// SIMATIC S7-200 project (STEP 7-Micro/WIN), CPU 226 REL 01.23

ORGANIZATION_BLOCK MAIN:OB1
TITLE= 
// PROGRAM COMMENTS
// Press F1 for help and example program
//  
BEGIN
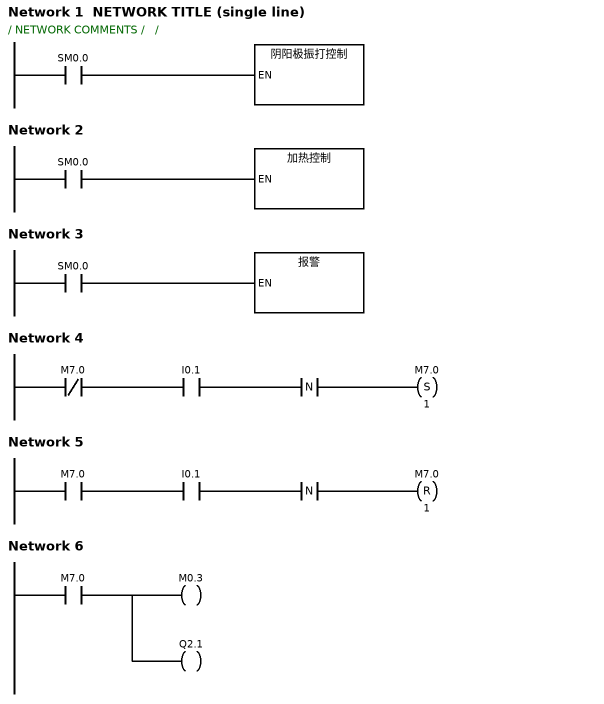
Network 1 // NETWORK TITLE (single line)
//  
// NETWORK COMMENTS
//  
// 
LD     SM0.0
CALL   阴阳极振打控制:SBR0
Network 2
LD     SM0.0
CALL   加热控制:SBR1
Network 3
LD     SM0.0
CALL   报警:SBR2
Network 4
LDN    M7.0
A      I0.1
ED
S      M7.0, 1
Network 5
LD     M7.0
A      I0.1
ED
R      M7.0, 1
Network 6
LD     M7.0
=      M0.3
=      Q2.1
END_ORGANIZATION_BLOCK

SUBROUTINE_BLOCK 阴阳极振打控制:SBR0
TITLE= 
// SUBROUTINE COMMENTS
// Press F1 for help and example program
//  
BEGIN
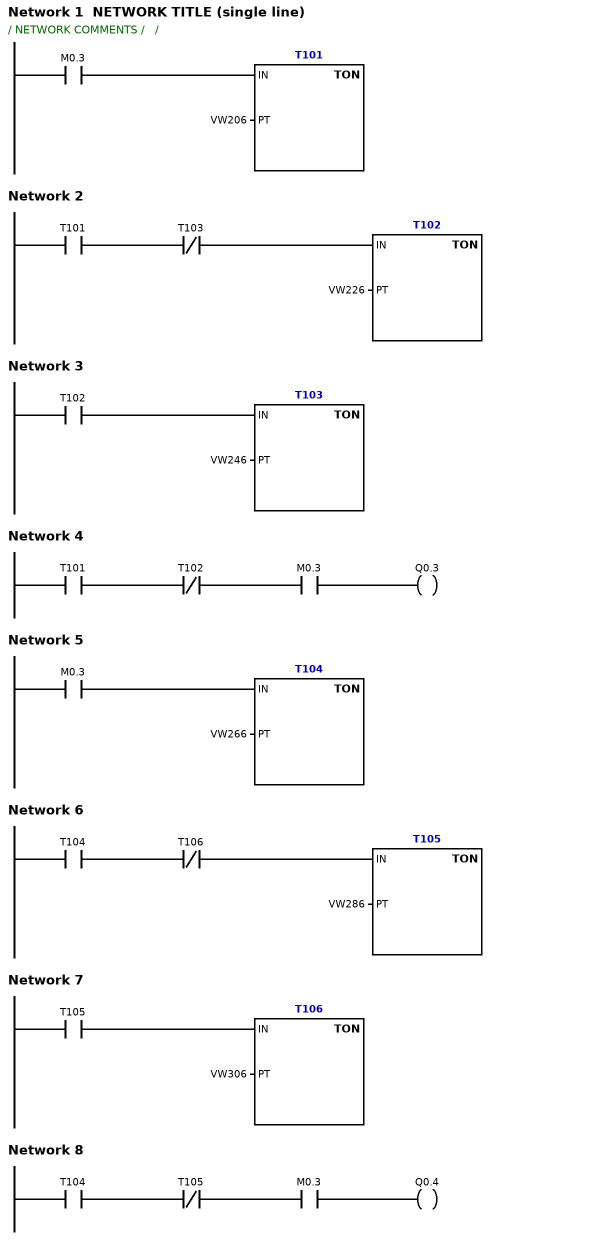
Network 1 // NETWORK TITLE (single line)
//  
// NETWORK COMMENTS
//  
// 
LD     M0.3
TON    T101, VW206
Network 2
LD     T101
AN     T103
TON    T102, VW226
Network 3
LD     T102
TON    T103, VW246
Network 4
LD     T101
AN     T102
A      M0.3
=      Q0.3
Network 5
LD     M0.3
TON    T104, VW266
Network 6
LD     T104
AN     T106
TON    T105, VW286
Network 7
LD     T105
TON    T106, VW306
Network 8
LD     T104
AN     T105
A      M0.3
=      Q0.4
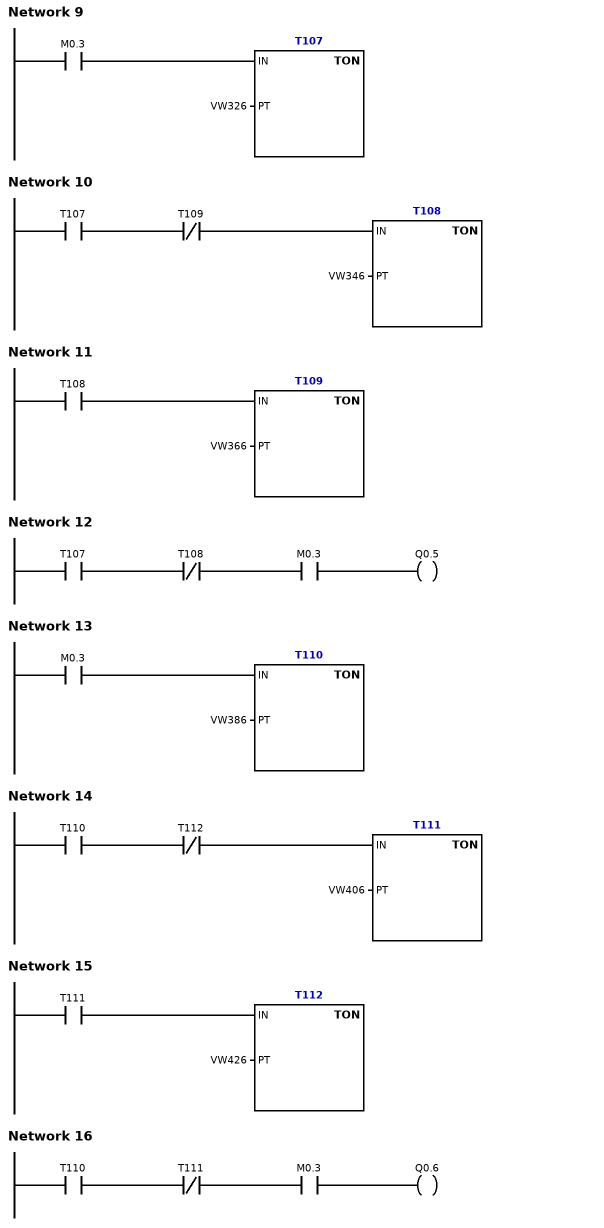
Network 9
LD     M0.3
TON    T107, VW326
Network 10
LD     T107
AN     T109
TON    T108, VW346
Network 11
LD     T108
TON    T109, VW366
Network 12
LD     T107
AN     T108
A      M0.3
=      Q0.5
Network 13
LD     M0.3
TON    T110, VW386
Network 14
LD     T110
AN     T112
TON    T111, VW406
Network 15
LD     T111
TON    T112, VW426
Network 16
LD     T110
AN     T111
A      M0.3
=      Q0.6
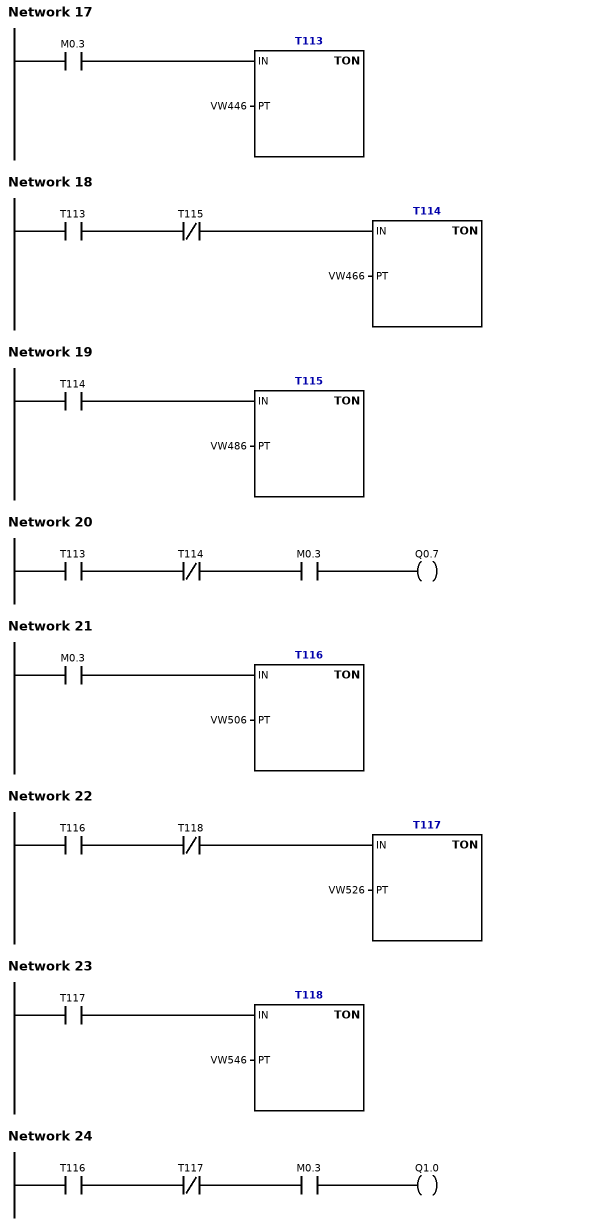
Network 17
LD     M0.3
TON    T113, VW446
Network 18
LD     T113
AN     T115
TON    T114, VW466
Network 19
LD     T114
TON    T115, VW486
Network 20
LD     T113
AN     T114
A      M0.3
=      Q0.7
Network 21
LD     M0.3
TON    T116, VW506
Network 22
LD     T116
AN     T118
TON    T117, VW526
Network 23
LD     T117
TON    T118, VW546
Network 24
LD     T116
AN     T117
A      M0.3
=      Q1.0
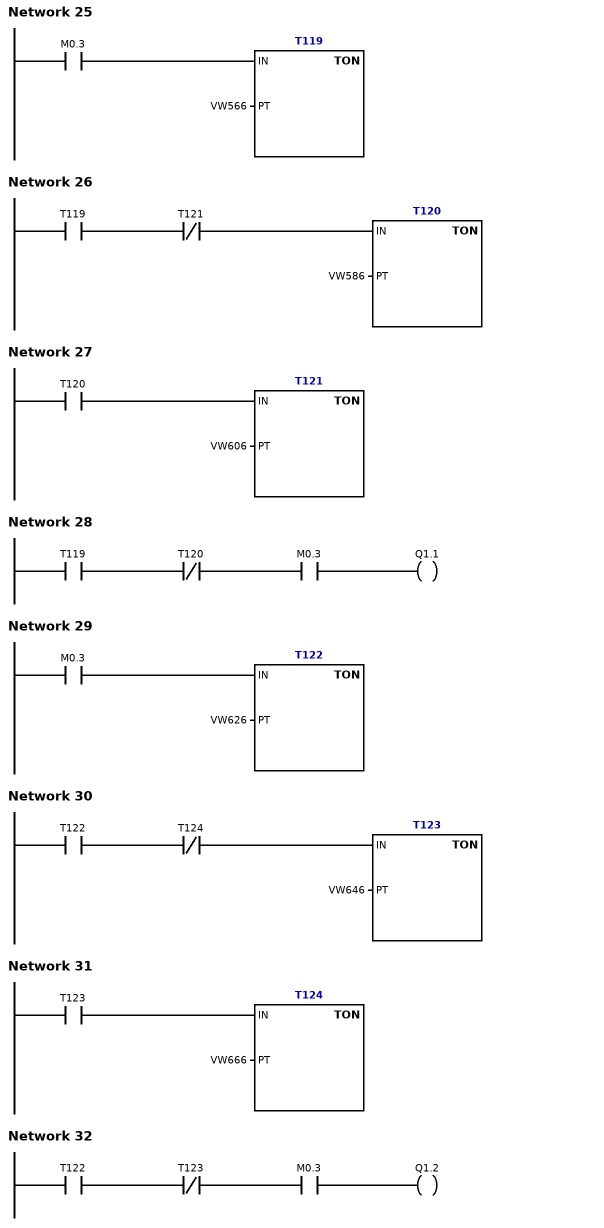
Network 25
LD     M0.3
TON    T119, VW566
Network 26
LD     T119
AN     T121
TON    T120, VW586
Network 27
LD     T120
TON    T121, VW606
Network 28
LD     T119
AN     T120
A      M0.3
=      Q1.1
Network 29
LD     M0.3
TON    T122, VW626
Network 30
LD     T122
AN     T124
TON    T123, VW646
Network 31
LD     T123
TON    T124, VW666
Network 32
LD     T122
AN     T123
A      M0.3
=      Q1.2
END_SUBROUTINE_BLOCK

SUBROUTINE_BLOCK 加热控制:SBR1
TITLE=
BEGIN
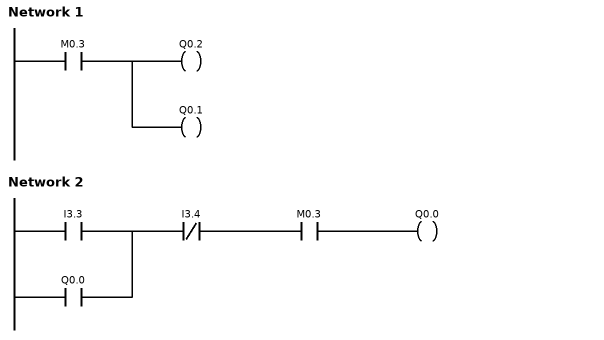
Network 1
LD     M0.3
=      Q0.2
=      Q0.1
Network 2
LD     I3.3
O      Q0.0
AN     I3.4
A      M0.3
=      Q0.0
END_SUBROUTINE_BLOCK

SUBROUTINE_BLOCK 报警:SBR2
TITLE=
BEGIN
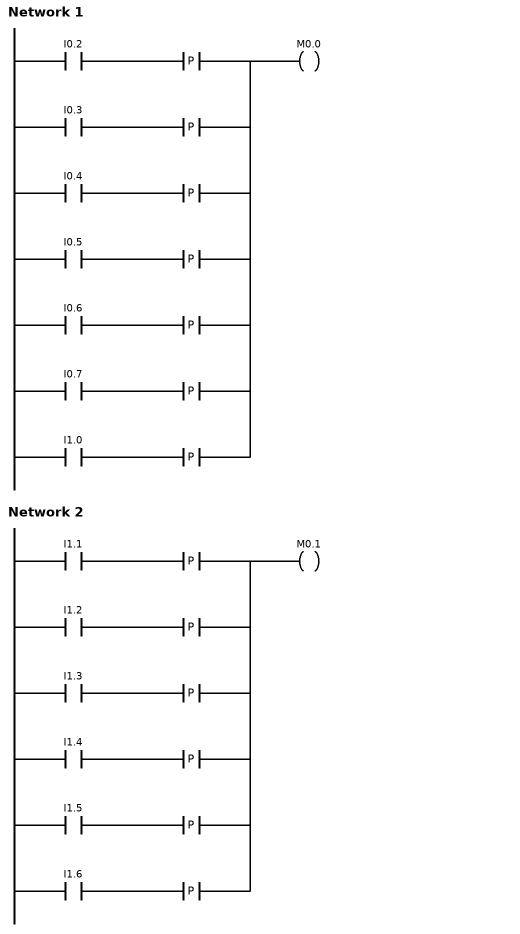
Network 1
LD     I0.2
EU
LD     I0.3
EU
OLD
LD     I0.4
EU
OLD
LD     I0.5
EU
OLD
LD     I0.6
EU
OLD
LD     I0.7
EU
OLD
LD     I1.0
EU
OLD
=      M0.0
Network 2
LD     I1.1
EU
LD     I1.2
EU
OLD
LD     I1.3
EU
OLD
LD     I1.4
EU
OLD
LD     I1.5
EU
OLD
LD     I1.6
EU
OLD
=      M0.1
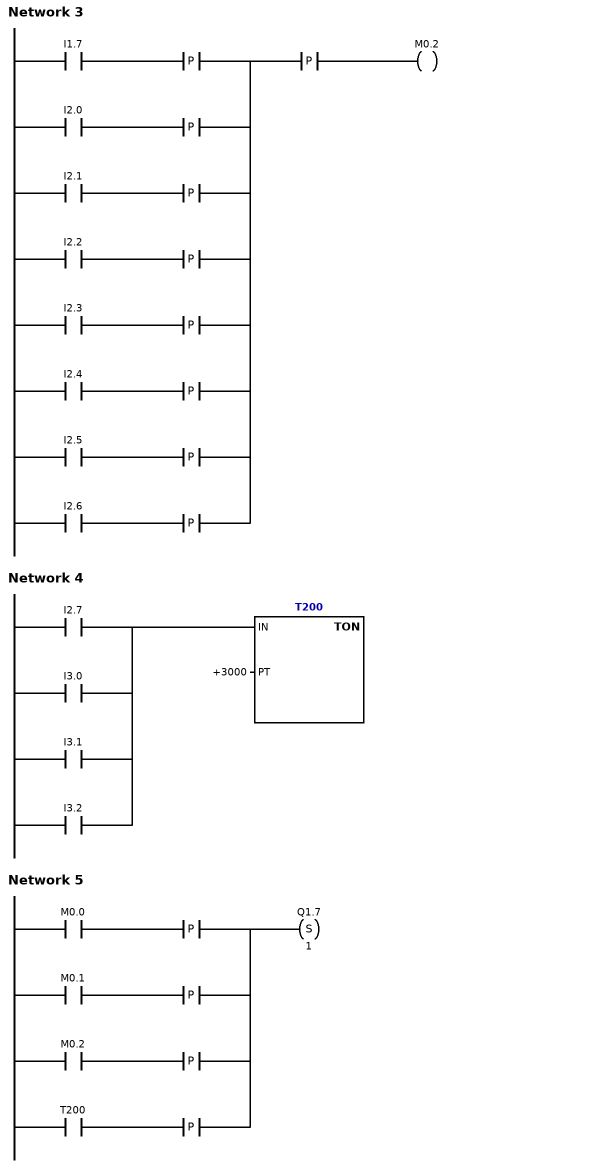
Network 3
LD     I1.7
EU
LD     I2.0
EU
OLD
LD     I2.1
EU
OLD
LD     I2.2
EU
OLD
LD     I2.3
EU
OLD
LD     I2.4
EU
OLD
LD     I2.5
EU
OLD
LD     I2.6
EU
OLD
EU
=      M0.2
Network 4
LD     I2.7
O      I3.0
O      I3.1
O      I3.2
TON    T200, +3000
Network 5
LD     M0.0
EU
LD     M0.1
EU
OLD
LD     M0.2
EU
OLD
LD     T200
EU
OLD
S      Q1.7, 1
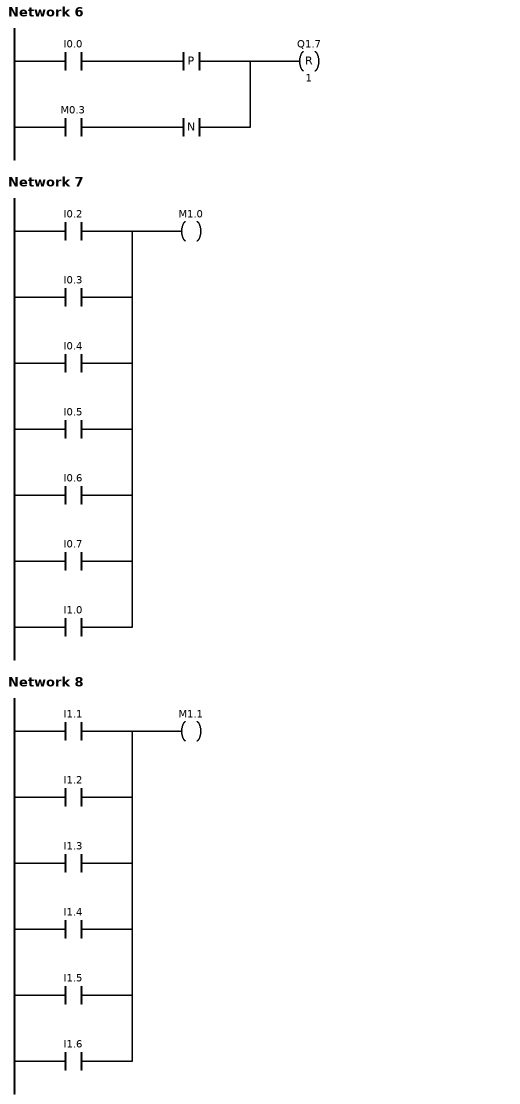
Network 6
LD     I0.0
EU
LD     M0.3
ED
OLD
R      Q1.7, 1
Network 7
LD     I0.2
O      I0.3
O      I0.4
O      I0.5
O      I0.6
O      I0.7
O      I1.0
=      M1.0
Network 8
LD     I1.1
O      I1.2
O      I1.3
O      I1.4
O      I1.5
O      I1.6
=      M1.1
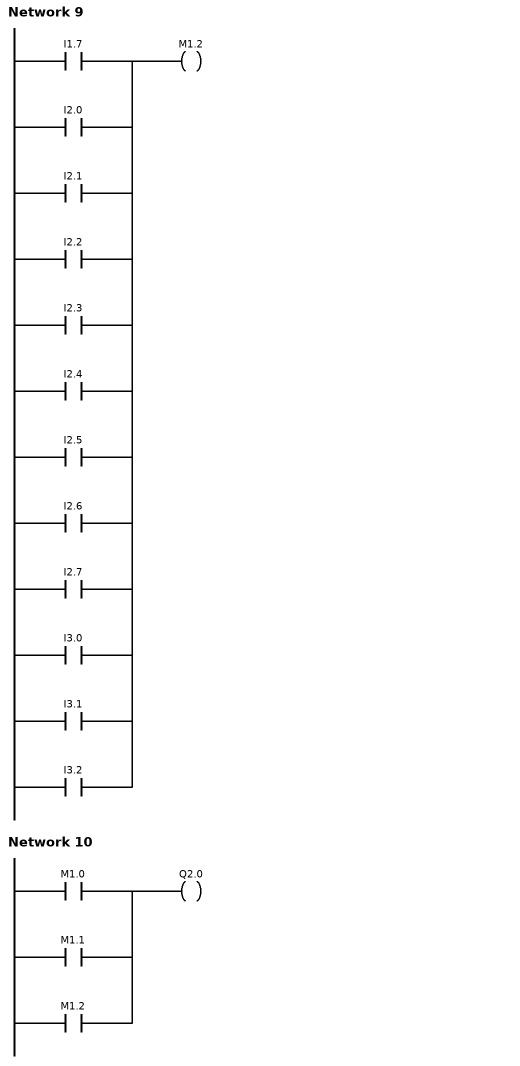
Network 9
LD     I1.7
O      I2.0
O      I2.1
O      I2.2
O      I2.3
O      I2.4
O      I2.5
O      I2.6
O      I2.7
O      I3.0
O      I3.1
O      I3.2
=      M1.2
Network 10
LD     M1.0
O      M1.1
O      M1.2
=      Q2.0
END_SUBROUTINE_BLOCK

DATA_BLOCK_TAB 用户定义1
BEGIN
VB0      16#0
VB1      16#0
VB2      16#0
VB3      16#0
VB4      16#0
VB5      16#0
VB6      16#0
VB7      16#0
VB8      16#0
VB9      16#0
VB10     16#0
VB11     16#0
VB12     16#0
VB13     16#0
VB14     16#0
VB15     16#0
VB16     16#0
VB17     16#0
VB18     16#0
VB19     16#0
VB20     16#0
VB21     16#0
VB22     16#0
VB23     16#0
VB24     16#0
VB25     16#0
VB26     16#0
VB27     16#0
VB28     16#0
VB29     16#0
VB30     16#0
VB31     16#0
VB32     16#0
VB33     16#0
VB34     16#0
VB35     16#0
VB36     16#0
VB37     16#0
VB38     16#0
VB39     16#0
VB40     16#0
VB41     16#0
VB42     16#0
VB43     16#0
VB44     16#0
VB45     16#0
VB46     16#0
VB47     16#0
VB48     16#0
VB49     16#0
VB50     16#0
VB51     16#0
VB52     16#0
VB53     16#0
VB54     16#0
VB55     16#0
VB56     16#0
VB57     16#0
VB58     16#0
VB59     16#0
VB60     16#0
VB61     16#0
VB62     16#0
VB63     16#0
VB64     16#0
VB65     16#0
VB66     16#0
VB67     16#0
VB68     16#0
VB69     16#0
VB70     16#0
VB71     16#0
VB72     16#0
VB73     16#0
VB74     16#0
VB75     16#0
VB76     16#0
VB77     16#0
VB78     16#0
VB79     16#0
VB80     16#0
VB81     16#0
VB82     16#0
VB83     16#0
VB84     16#0
VB85     16#0
VB86     16#0
VB87     16#0
VB88     16#0
VB89     16#0
VB90     16#0
VB91     16#0
VB92     16#0
VB93     16#0
VB94     16#0
VB95     16#0
VB96     16#0
VB97     16#0
VB98     16#0
VB99     16#0
VB100    16#0
VB101    16#0
VB102    16#0
VB103    16#0
VB104    16#0
VB105    16#0
VB106    16#0
VB107    16#0
VB108    16#0
VB109    16#0
VB110    16#0
VB111    16#0
VB112    16#0
VB113    16#0
VB114    16#0
VB115    16#0
VB116    16#0
VB117    16#0
VB118    16#0
VB119    16#0
VB120    16#0
VB121    16#0
VB122    16#0
VB123    16#0
VB124    16#0
VB125    16#0
VB126    16#0
VB127    16#0
VB128    16#0
VB129    16#0
VB130    16#0
VB131    16#0
VB132    16#0
VB133    16#0
VB134    16#0
VB135    16#0
VB136    16#0
VB137    16#0
VB138    16#0
VB139    16#0
VB140    16#0
VB141    16#0
VB142    16#0
VB143    16#0
VB144    16#0
VB145    16#0
VB146    16#0
VB147    16#0
VB148    16#0
VB149    16#0
VB150    16#0
VB151    16#0
VB152    16#0
VB153    16#0
VB154    16#0
VB155    16#0
VB156    16#0
VB157    16#0
VB158    16#0
VB159    16#0
VB160    16#0
VB161    16#0
VB162    16#0
VB163    16#0
VB164    16#0
VB165    16#0
VB166    16#0
VB167    16#0
VB168    16#0
VB169    16#0
VB170    16#0
VB171    16#0
VB172    16#0
VB173    16#0
VB174    16#0
VB175    16#0
VB176    16#0
VB177    16#0
VB178    16#0
VB179    16#0
VB180    16#0
VB181    16#0
VB182    16#0
VB183    16#0
VB184    16#0
VB185    16#0
VB186    16#0
VB187    16#0
VB188    16#0
VB189    16#0
VB190    16#0
VB191    16#0
VB192    16#0
VB193    16#0
VB194    16#0
VB195    16#0
VB196    16#0
VB197    16#0
VB198    16#0
VB199    16#0
VB200    16#0
VB201    16#0
VB202    16#0
VB203    16#0
VB204    16#0
VB205    16#0
VB206    16#0
VB207    16#0
VB208    16#0
VB209    16#0
VB210    16#0
VB211    16#0
VB212    16#0
VB213    16#0
VB214    16#0
VB215    16#0
VB216    16#0
VB217    16#0
VB218    16#0
VB219    16#0
VB220    16#0
VB221    16#0
VB222    16#0
VB223    16#0
VB224    16#0
VB225    16#0
VB226    16#5
VB227    16#DC
VB228    16#0
VB229    16#0
VB230    16#0
VB231    16#0
VB232    16#0
VB233    16#0
VB234    16#0
VB235    16#0
VB236    16#0
VB237    16#0
VB238    16#0
VB239    16#0
VB240    16#0
VB241    16#0
VB242    16#0
VB243    16#0
VB244    16#0
VB245    16#0
VB246    16#5
VB247    16#DC
VB248    16#0
VB249    16#0
VB250    16#0
VB251    16#0
VB252    16#0
VB253    16#0
VB254    16#0
VB255    16#0
VB256    16#0
VB257    16#0
VB258    16#0
VB259    16#0
VB260    16#0
VB261    16#0
VB262    16#0
VB263    16#0
VB264    16#0
VB265    16#0
VB266    16#5
VB267    16#DC
VB268    16#0
VB269    16#0
VB270    16#0
VB271    16#0
VB272    16#0
VB273    16#0
VB274    16#0
VB275    16#0
VB276    16#0
VB277    16#0
VB278    16#0
VB279    16#0
VB280    16#0
VB281    16#0
VB282    16#0
VB283    16#0
VB284    16#0
VB285    16#0
VB286    16#5
VB287    16#DC
VB288    16#0
VB289    16#0
VB290    16#0
VB291    16#0
VB292    16#0
VB293    16#0
VB294    16#0
VB295    16#0
VB296    16#0
VB297    16#0
VB298    16#0
VB299    16#0
VB300    16#0
VB301    16#0
VB302    16#0
VB303    16#0
VB304    16#0
VB305    16#0
VB306    16#11
VB307    16#94
VB308    16#0
VB309    16#0
VB310    16#0
VB311    16#0
VB312    16#0
VB313    16#0
VB314    16#0
VB315    16#0
VB316    16#0
VB317    16#0
VB318    16#0
VB319    16#0
VB320    16#0
VB321    16#0
VB322    16#0
VB323    16#0
VB324    16#0
VB325    16#0
VB326    16#11
VB327    16#94
VB328    16#0
VB329    16#0
VB330    16#0
VB331    16#0
VB332    16#0
VB333    16#0
VB334    16#0
VB335    16#0
VB336    16#0
VB337    16#0
VB338    16#0
VB339    16#0
VB340    16#0
VB341    16#0
VB342    16#0
VB343    16#0
VB344    16#0
VB345    16#0
VB346    16#5
VB347    16#DC
VB348    16#0
VB349    16#0
VB350    16#0
VB351    16#0
VB352    16#0
VB353    16#0
VB354    16#0
VB355    16#0
VB356    16#0
VB357    16#0
VB358    16#0
VB359    16#0
VB360    16#0
VB361    16#0
VB362    16#0
VB363    16#0
VB364    16#0
VB365    16#0
VB366    16#29
VB367    16#4
VB368    16#0
VB369    16#0
VB370    16#0
VB371    16#0
VB372    16#0
VB373    16#0
VB374    16#0
VB375    16#0
VB376    16#0
VB377    16#0
VB378    16#0
VB379    16#0
VB380    16#0
VB381    16#0
VB382    16#0
VB383    16#0
VB384    16#0
VB385    16#0
VB386    16#17
VB387    16#70
VB388    16#0
VB389    16#0
VB390    16#0
VB391    16#0
VB392    16#0
VB393    16#0
VB394    16#0
VB395    16#0
VB396    16#0
VB397    16#0
VB398    16#0
VB399    16#0
VB400    16#0
VB401    16#0
VB402    16#0
VB403    16#0
VB404    16#0
VB405    16#0
VB406    16#5
VB407    16#DC
VB408    16#0
VB409    16#0
VB410    16#0
VB411    16#0
VB412    16#0
VB413    16#0
VB414    16#0
VB415    16#0
VB416    16#0
VB417    16#0
VB418    16#0
VB419    16#0
VB420    16#0
VB421    16#0
VB422    16#0
VB423    16#0
VB424    16#0
VB425    16#0
VB426    16#40
VB427    16#74
VB428    16#0
VB429    16#0
VB430    16#0
VB431    16#0
VB432    16#0
VB433    16#0
VB434    16#0
VB435    16#0
VB436    16#0
VB437    16#0
VB438    16#0
VB439    16#0
VB440    16#0
VB441    16#0
VB442    16#0
VB443    16#0
VB444    16#0
VB445    16#0
VB446    16#5
VB447    16#DC
VB448    16#0
VB449    16#0
VB450    16#0
VB451    16#0
VB452    16#0
VB453    16#0
VB454    16#0
VB455    16#0
VB456    16#0
VB457    16#0
VB458    16#0
VB459    16#0
VB460    16#0
VB461    16#0
VB462    16#0
VB463    16#0
VB464    16#0
VB465    16#0
VB466    16#5
VB467    16#DC
VB468    16#0
VB469    16#0
VB470    16#0
VB471    16#0
VB472    16#0
VB473    16#0
VB474    16#0
VB475    16#0
VB476    16#0
VB477    16#0
VB478    16#0
VB479    16#0
VB480    16#0
VB481    16#0
VB482    16#0
VB483    16#0
VB484    16#0
VB485    16#0
VB486    16#5
VB487    16#DC
VB488    16#0
VB489    16#0
VB490    16#0
VB491    16#0
VB492    16#0
VB493    16#0
VB494    16#0
VB495    16#0
VB496    16#0
VB497    16#0
VB498    16#0
VB499    16#0
VB500    16#0
VB501    16#0
VB502    16#0
VB503    16#0
VB504    16#0
VB505    16#0
VB506    16#B
VB507    16#B8
VB508    16#0
VB509    16#0
VB510    16#0
VB511    16#0
VB512    16#0
VB513    16#0
VB514    16#0
VB515    16#0
VB516    16#0
VB517    16#0
VB518    16#0
VB519    16#0
VB520    16#0
VB521    16#0
VB522    16#0
VB523    16#0
VB524    16#0
VB525    16#0
VB526    16#5
VB527    16#DC
VB528    16#0
VB529    16#0
VB530    16#0
VB531    16#0
VB532    16#0
VB533    16#0
VB534    16#0
VB535    16#0
VB536    16#0
VB537    16#0
VB538    16#0
VB539    16#0
VB540    16#0
VB541    16#0
VB542    16#0
VB543    16#0
VB544    16#0
VB545    16#0
VB546    16#5
VB547    16#DC
VB548    16#0
VB549    16#0
VB550    16#0
VB551    16#0
VB552    16#0
VB553    16#0
VB554    16#0
VB555    16#0
VB556    16#0
VB557    16#0
VB558    16#0
VB559    16#0
VB560    16#0
VB561    16#0
VB562    16#0
VB563    16#0
VB564    16#0
VB565    16#0
VB566    16#11
VB567    16#94
VB568    16#0
VB569    16#0
VB570    16#0
VB571    16#0
VB572    16#0
VB573    16#0
VB574    16#0
VB575    16#0
VB576    16#0
VB577    16#0
VB578    16#0
VB579    16#0
VB580    16#0
VB581    16#0
VB582    16#0
VB583    16#0
VB584    16#0
VB585    16#0
VB586    16#5
VB587    16#DC
VB588    16#0
VB589    16#0
VB590    16#0
VB591    16#0
VB592    16#0
VB593    16#0
VB594    16#0
VB595    16#0
VB596    16#0
VB597    16#0
VB598    16#0
VB599    16#0
VB600    16#0
VB601    16#0
VB602    16#0
VB603    16#0
VB604    16#0
VB605    16#0
VB606    16#5
VB607    16#DC
VB608    16#0
VB609    16#0
VB610    16#0
VB611    16#0
VB612    16#0
VB613    16#0
VB614    16#0
VB615    16#0
VB616    16#0
VB617    16#0
VB618    16#0
VB619    16#0
VB620    16#0
VB621    16#0
VB622    16#0
VB623    16#0
VB624    16#0
VB625    16#0
VB626    16#17
VB627    16#70
VB628    16#0
VB629    16#0
VB630    16#0
VB631    16#0
VB632    16#0
VB633    16#0
VB634    16#0
VB635    16#0
VB636    16#0
VB637    16#0
VB638    16#0
VB639    16#0
VB640    16#0
VB641    16#0
VB642    16#0
VB643    16#0
VB644    16#0
VB645    16#0
VB646    16#5
VB647    16#DC
VB648    16#0
VB649    16#0
VB650    16#0
VB651    16#0
VB652    16#0
VB653    16#0
VB654    16#0
VB655    16#0
VB656    16#0
VB657    16#0
VB658    16#0
VB659    16#0
VB660    16#0
VB661    16#0
VB662    16#0
VB663    16#0
VB664    16#0
VB665    16#0
VB666    16#5
VB667    16#DC
VB668    16#0
VB669    16#0
VB670    16#0
VB671    16#0
VB672    16#0
VB673    16#0
VB674    16#0
VB675    16#0
VB676    16#0
VB677    16#0
VB678    16#0
VB679    16#0
VB680    16#0
VB681    16#0
VB682    16#0
VB683    16#0
VB684    16#0
VB685    16#0
VB686    16#B
VB687    16#B8
VB688    16#0
VB689    16#0
VB690    16#0
VB691    16#0
VB692    16#0
VB693    16#0
VB694    16#0
VB695    16#0
VB696    16#0
VB697    16#0
VB698    16#0
VB699    16#0
VB700    16#0
VB701    16#0
VB702    16#0
VB703    16#0
VB704    16#0
VB705    16#0
VB706    16#B
VB707    16#B8
VB708    16#0
VB709    16#0
VB710    16#0
VB711    16#0
VB712    16#0
VB713    16#0
VB714    16#0
VB715    16#0
VB716    16#0
VB717    16#0
VB718    16#0
VB719    16#0
VB720    16#0
VB721    16#0
VB722    16#0
VB723    16#0
VB724    16#0
VB725    16#0
VB726    16#B
VB727    16#B8
VB728    16#0
VB729    16#0
VB730    16#0
VB731    16#0
VB732    16#0
VB733    16#0
VB734    16#0
VB735    16#0
VB736    16#0
VB737    16#0
VB738    16#0
VB739    16#0
VB740    16#0
VB741    16#0
VB742    16#0
VB743    16#0
VB744    16#0
VB745    16#0
VB746    16#17
VB747    16#70
VB748    16#0
VB749    16#0
VB750    16#0
VB751    16#0
VB752    16#0
VB753    16#0
VB754    16#0
VB755    16#0
VB756    16#0
VB757    16#0
VB758    16#0
VB759    16#0
VB760    16#0
VB761    16#0
VB762    16#0
VB763    16#0
VB764    16#0
VB765    16#0
VB766    16#B
VB767    16#B8
VB768    16#0
VB769    16#0
VB770    16#0
VB771    16#0
VB772    16#0
VB773    16#0
VB774    16#0
VB775    16#0
VB776    16#0
VB777    16#0
VB778    16#0
VB779    16#0
VB780    16#0
VB781    16#0
VB782    16#0
VB783    16#0
VB784    16#0
VB785    16#0
VB786    16#17
VB787    16#70
VB788    16#0
VB789    16#0
VB790    16#0
VB791    16#0
VB792    16#0
VB793    16#0
VB794    16#0
VB795    16#0
VB796    16#0
VB797    16#0
VB798    16#0
VB799    16#0
VB800    16#0
VB801    16#0
VB802    16#0
VB803    16#0
VB804    16#0
VB805    16#0
VB806    16#23
VB807    16#28
VB808    16#0
VB809    16#0
VB810    16#0
VB811    16#0
VB812    16#0
VB813    16#0
VB814    16#0
VB815    16#0
VB816    16#0
VB817    16#0
VB818    16#0
VB819    16#0
VB820    16#0
VB821    16#0
VB822    16#0
VB823    16#0
VB824    16#0
VB825    16#0
VB826    16#B
VB827    16#B8
VB828    16#0
VB829    16#0
VB830    16#0
VB831    16#0
VB832    16#0
VB833    16#0
VB834    16#0
VB835    16#0
VB836    16#0
VB837    16#0
VB838    16#0
VB839    16#0
VB840    16#0
VB841    16#0
VB842    16#0
VB843    16#0
VB844    16#0
VB845    16#0
VB846    16#23
VB847    16#28
VB848    16#0
VB849    16#0
VB850    16#0
VB851    16#0
VB852    16#0
VB853    16#0
VB854    16#0
VB855    16#0
VB856    16#0
VB857    16#0
VB858    16#0
VB859    16#0
VB860    16#0
VB861    16#0
VB862    16#0
VB863    16#0
VB864    16#0
VB865    16#0
VB866    16#2E
VB867    16#E0
VB868    16#0
VB869    16#0
VB870    16#0
VB871    16#0
VB872    16#0
VB873    16#0
VB874    16#0
VB875    16#0
VB876    16#0
VB877    16#0
VB878    16#0
VB879    16#0
VB880    16#0
VB881    16#0
VB882    16#0
VB883    16#0
VB884    16#0
VB885    16#0
VB886    16#B
VB887    16#B8
VB888    16#0
VB889    16#0
VB890    16#0
VB891    16#0
VB892    16#0
VB893    16#0
VB894    16#0
VB895    16#0
VB896    16#0
VB897    16#0
VB898    16#0
VB899    16#0
VB900    16#0
VB901    16#0
VB902    16#0
VB903    16#0
VB904    16#0
VB905    16#0
VB906    16#3A
VB907    16#98
END_DATA_BLOCK_TAB
